FUNCTION_BLOCK booleanAssertionTests EXTENDS FB_TestSuite

VAR
	concrete	: IAssertionTestable;
END_VAR

testBoolIsTrue();
testBoolIsFalse();
testBoolIsEqual();
testBoolIsNotEqual();

METHOD FB_init : BOOL
VAR_INPUT
    bInitRetains : BOOL; // if TRUE, the retain variables are initialized (warm start / cold start)
    bInCopyCode : BOOL;  // if TRUE, the instance afterwards gets moved into the copy code (online change)
	concrete : IAssertionTestable;
END_VAR
THIS^.concrete := concrete;
END_METHOD

METHOD reset
VAR_INPUT
END_VAR
THIS^.concrete.assertionWasWrong  := FALSE;
END_METHOD

METHOD testBoolIsEqual

VAR
	testVarCurrent : BOOL;
	testVarExpected : BOOL;
END_VAR
TEST('Boolean is EqualTo' );

// Test Number 0
THIS^.reset();
THIS^.concrete.assert.boolean.valueIsEqualTo(
	currentValue 	:= testVarCurrent,
	expectedValue	:= testVarExpected,
	message			:= ''
);

THIS^.AssertEquals_BOOL(
	Expected 	:= FALSE,
	Actual 		:= THIS^.concrete.assertionWasWrong,
	Message 	:= 'Test number 0 for boolean.isEqualTo assertion failed'
);

// Test Number 1
THIS^.reset();
testVarCurrent := TRUE;
THIS^.concrete.assert.boolean.valueIsEqualTo(
	currentValue 	:= testVarCurrent,
	expectedValue	:= testVarExpected,
	message			:= ''
);

THIS^.AssertEquals_BOOL(
	Expected 	:= TRUE,
	Actual 		:= THIS^.concrete.assertionWasWrong,
	Message 	:= 'Test number 1 for boolean.isEqualTo assertion failed'
);

// Test Number 2
THIS^.reset();
testVarCurrent := FALSE;
testVarExpected := TRUE;
THIS^.concrete.assert.boolean.valueIsEqualTo(
	currentValue 	:= testVarCurrent,
	expectedValue	:= testVarExpected,
	message			:= ''
);

THIS^.AssertEquals_BOOL(
	Expected 	:= TRUE,
	Actual 		:= THIS^.concrete.assertionWasWrong,
	Message 	:= 'Test number 2 for boolean.isEqualTo assertion failed'
);

// Test Number 3
THIS^.reset();
testVarCurrent := TRUE;
testVarExpected := FALSE;
THIS^.concrete.assert.boolean.valueIsEqualTo(
	currentValue 	:= testVarCurrent,
	expectedValue	:= testVarExpected,
	message			:= ''
);

THIS^.AssertEquals_BOOL(
	Expected 	:= TRUE,
	Actual 		:= THIS^.concrete.assertionWasWrong,
	Message 	:= 'Test number 3 for boolean.isEqualTo assertion failed'
);

// Test Number 4
THIS^.reset();
testVarCurrent := TRUE;
testVarExpected := 0;
THIS^.concrete.assert.boolean.valueIsEqualTo(
	currentValue 	:= testVarCurrent,
	expectedValue	:= testVarExpected,
	message			:= ''
);

THIS^.AssertEquals_BOOL(
	Expected 	:= TRUE,
	Actual 		:= THIS^.concrete.assertionWasWrong,
	Message 	:= 'Test number 4 for boolean.isEqualTo assertion failed'
);

// Test Number 5
THIS^.reset();
testVarCurrent := 1;
testVarExpected := 0;
THIS^.concrete.assert.boolean.valueIsEqualTo(
	currentValue 	:= testVarCurrent,
	expectedValue	:= testVarExpected,
	message			:= ''
);

THIS^.AssertEquals_BOOL(
	Expected 	:= TRUE,
	Actual 		:= THIS^.concrete.assertionWasWrong,
	Message 	:= 'Test number 5 for boolean.isEqualTo assertion failed'
);

// Test Number 6
THIS^.reset();
testVarCurrent := 1;
testVarExpected := 1;
THIS^.concrete.assert.boolean.valueIsEqualTo(
	currentValue 	:= testVarCurrent,
	expectedValue	:= testVarExpected,
	message			:= ''
);

THIS^.AssertEquals_BOOL(
	Expected 	:= FALSE,
	Actual 		:= THIS^.concrete.assertionWasWrong,
	Message 	:= 'Test number 6 for boolean.isEqualTo assertion failed'
);

// Test Number 7
THIS^.reset();
testVarCurrent := 0;
testVarExpected := 0;
THIS^.concrete.assert.boolean.valueIsEqualTo(
	currentValue 	:= testVarCurrent,
	expectedValue	:= testVarExpected,
	message			:= ''
);

THIS^.AssertEquals_BOOL(
	Expected 	:= FALSE,
	Actual 		:= THIS^.concrete.assertionWasWrong,
	Message 	:= 'Test number 7 for boolean.isEqualTo assertion failed'
);

// Test Number 8
THIS^.reset();
testVarCurrent := TRUE;
testVarExpected := TRUE;
THIS^.concrete.assert.boolean.valueIsEqualTo(
	currentValue 	:= testVarCurrent,
	expectedValue	:= testVarExpected,
	message			:= ''
);

THIS^.AssertEquals_BOOL(
	Expected 	:= FALSE,
	Actual 		:= THIS^.concrete.assertionWasWrong,
	Message 	:= 'Test number 8 for boolean.isEqualTo assertion failed'
);

// Test Number 9
THIS^.reset();
testVarCurrent := FALSE;
testVarExpected := FALSE;
THIS^.concrete.assert.boolean.valueIsEqualTo(
	currentValue 	:= testVarCurrent,
	expectedValue	:= testVarExpected,
	message			:= ''
);

THIS^.AssertEquals_BOOL(
	Expected 	:= FALSE,
	Actual 		:= THIS^.concrete.assertionWasWrong,
	Message 	:= 'Test number 9 for boolean.isEqualTo assertion failed'
);

TEST_FINISHED();
END_METHOD

METHOD testBoolIsFalse

VAR
	testBoolVar : BOOL;	
END_VAR
TEST('Boolean is False' );

// Test number 0
THIS^.reset();
THIS^.concrete.assert.boolean.valueIsFalse(
	currentValue 	:= testBoolVar,
	message			:= ''
);						

THIS^.AssertEquals_BOOL(
	Expected 	:= FALSE,
	Actual 		:= THIS^.concrete.assertionWasWrong,
	Message 	:= 'Test number 0 for boolean.isFalse assertion failed'
);

// Test number 1
THIS^.reset();
testBoolVar := TRUE;
THIS^.concrete.assert.boolean.valueIsFalse(
	currentValue 	:= testBoolVar,
	message			:= ''
);						

THIS^.AssertEquals_BOOL(
	Expected 	:= TRUE,
	Actual 		:= THIS^.concrete.assertionWasWrong,
	Message 	:= 'Test number 1 for boolean.isFalse assertion failed'
);

// Test number 2
THIS^.reset();
testBoolVar := FALSE;
THIS^.concrete.assert.boolean.valueIsFalse(
	currentValue 	:= testBoolVar,
	message			:= ''
);						

THIS^.AssertEquals_BOOL(
	Expected 	:= FALSE,
	Actual 		:= THIS^.concrete.assertionWasWrong,
	Message 	:= 'Test number 2 for boolean.isFalse assertion failed'
);

// Test number 3
THIS^.reset();
testBoolVar := 0;
THIS^.concrete.assert.boolean.valueIsFalse(
	currentValue 	:= testBoolVar,
	message			:= ''
);						

THIS^.AssertEquals_BOOL(
	Expected 	:= FALSE,
	Actual 		:= THIS^.concrete.assertionWasWrong,
	Message 	:= 'Test number 3 for boolean.isFalse assertion failed'
);

// Test number 4
THIS^.reset();
testBoolVar := 1;
THIS^.concrete.assert.boolean.valueIsFalse(
	currentValue 	:= testBoolVar,
	message			:= ''
);						

THIS^.AssertEquals_BOOL(
	Expected 	:= TRUE,
	Actual 		:= THIS^.concrete.assertionWasWrong,
	Message 	:= 'Test number 4 for boolean.isFalse assertion failed'
);
TEST_FINISHED();
END_METHOD

METHOD testBoolIsNotEqual

VAR
	testVarCurrent : BOOL;
	testVarExpected : BOOL;
END_VAR
TEST('Boolean is NotEqualTo' );

// Test Number 0
THIS^.reset();
THIS^.concrete.assert.boolean.valueIsNotEqualTo(
	currentValue 	:= testVarCurrent,
	unexpectedValue	:= testVarExpected,
	message			:= ''
);

THIS^.AssertEquals_BOOL(
	Expected 	:= TRUE,
	Actual 		:= THIS^.concrete.assertionWasWrong,
	Message 	:= 'Test number 0 for boolean.notEqualTo assertion failed'
);

// Test Number 1
THIS^.reset();
testVarCurrent := TRUE;
THIS^.concrete.assert.boolean.valueIsNotEqualTo(
	currentValue 	:= testVarCurrent,
	unexpectedValue	:= testVarExpected,
	message			:= ''
);

THIS^.AssertEquals_BOOL(
	Expected 	:= FALSE,
	Actual 		:= THIS^.concrete.assertionWasWrong,
	Message 	:= 'Test number 1 for boolean.notEqualTo assertion failed'
);

// Test Number 2
THIS^.reset();
testVarCurrent := FALSE;
testVarExpected := TRUE;
THIS^.concrete.assert.boolean.valueIsNotEqualTo(
	currentValue 	:= testVarCurrent,
	unexpectedValue	:= testVarExpected,
	message			:= ''
);

THIS^.AssertEquals_BOOL(
	Expected 	:= FALSE,
	Actual 		:= THIS^.concrete.assertionWasWrong,
	Message 	:= 'Test number 2 for boolean.notEqualTo assertion failed'
);

// Test Number 3
THIS^.reset();
testVarCurrent := TRUE;
testVarExpected := FALSE;
THIS^.concrete.assert.boolean.valueIsNotEqualTo(
	currentValue 	:= testVarCurrent,
	unexpectedValue	:= testVarExpected,
	message			:= ''
);

THIS^.AssertEquals_BOOL(
	Expected 	:= FALSE,
	Actual 		:= THIS^.concrete.assertionWasWrong,
	Message 	:= 'Test number 3 for boolean.notEqualTo assertion failed'
);

// Test Number 4
THIS^.reset();
testVarCurrent := TRUE;
testVarExpected := 0;
THIS^.concrete.assert.boolean.valueIsNotEqualTo(
	currentValue 	:= testVarCurrent,
	unexpectedValue	:= testVarExpected,
	message			:= ''
);

THIS^.AssertEquals_BOOL(
	Expected 	:= FALSE,
	Actual 		:= THIS^.concrete.assertionWasWrong,
	Message 	:= 'Test number 4 for boolean.notEqualTo assertion failed'
);

// Test Number 5
THIS^.reset();
testVarCurrent := 1;
testVarExpected := 0;
THIS^.concrete.assert.boolean.valueIsNotEqualTo(
	currentValue 	:= testVarCurrent,
	unexpectedValue	:= testVarExpected,
	message			:= ''
);

THIS^.AssertEquals_BOOL(
	Expected 	:= FALSE,
	Actual 		:= THIS^.concrete.assertionWasWrong,
	Message 	:= 'Test number 5 for boolean.notEqualTo assertion failed'
);

// Test Number 6
THIS^.reset();
testVarCurrent := 1;
testVarExpected := 1;
THIS^.concrete.assert.boolean.valueIsNotEqualTo(
	currentValue 	:= testVarCurrent,
	unexpectedValue	:= testVarExpected,
	message			:= ''
);

THIS^.AssertEquals_BOOL(
	Expected 	:= TRUE,
	Actual 		:= THIS^.concrete.assertionWasWrong,
	Message 	:= 'Test number 6 for boolean.notEqualTo assertion failed'
);

// Test Number 7
THIS^.reset();
testVarCurrent := 0;
testVarExpected := 0;
THIS^.concrete.assert.boolean.valueIsNotEqualTo(
	currentValue 	:= testVarCurrent,
	unexpectedValue	:= testVarExpected,
	message			:= ''
);

THIS^.AssertEquals_BOOL(
	Expected 	:= TRUE,
	Actual 		:= THIS^.concrete.assertionWasWrong,
	Message 	:= 'Test number 7 for boolean.notEqualTo assertion failed'
);

// Test Number 8
THIS^.reset();
testVarCurrent := TRUE;
testVarExpected := TRUE;
THIS^.concrete.assert.boolean.valueIsNotEqualTo(
	currentValue 	:= testVarCurrent,
	unexpectedValue	:= testVarExpected,
	message			:= ''
);

THIS^.AssertEquals_BOOL(
	Expected 	:= TRUE,
	Actual 		:= THIS^.concrete.assertionWasWrong,
	Message 	:= 'Test number 8 for boolean.notEqualTo assertion failed'
);

// Test Number 9
THIS^.reset();
testVarCurrent := FALSE;
testVarExpected := FALSE;
THIS^.concrete.assert.boolean.valueIsNotEqualTo(
	currentValue 	:= testVarCurrent,
	unexpectedValue	:= testVarExpected,
	message			:= ''
);

THIS^.AssertEquals_BOOL(
	Expected 	:= TRUE,
	Actual 		:= THIS^.concrete.assertionWasWrong,
	Message 	:= 'Test number 9 for boolean.notEqualTo assertion failed'
);

TEST_FINISHED();
END_METHOD

METHOD testBoolIsTrue

VAR
	testBoolVar : BOOL;	
END_VAR
TEST('Boolean is true' );

// Test number 0
THIS^.reset();
THIS^.concrete.assert.boolean.valueIsTrue(
	currentValue 	:= testBoolVar,
	message			:= ''
);						

THIS^.AssertEquals_BOOL(
	Expected 	:= TRUE,
	Actual 		:= THIS^.concrete.assertionWasWrong,
	Message 	:= 'Test number 0 for boolean.isTrue assertion failed'
);

// Test number 1
THIS^.reset();
testBoolVar := TRUE;
THIS^.concrete.assert.boolean.valueIsTrue(
	currentValue 	:= testBoolVar,
	message			:= ''
);						

THIS^.AssertEquals_BOOL(
	Expected 	:= FALSE,
	Actual 		:= THIS^.concrete.assertionWasWrong,
	Message 	:= 'Test number 1 for boolean.isTrue assertion failed'
);

// Test number 2
THIS^.reset();
testBoolVar := FALSE;
THIS^.concrete.assert.boolean.valueIsTrue(
	currentValue 	:= testBoolVar,
	message			:= ''
);						

THIS^.AssertEquals_BOOL(
	Expected 	:= TRUE,
	Actual 		:= THIS^.concrete.assertionWasWrong,
	Message 	:= 'Test number 2 for boolean.isTrue assertion failed'
);

// Test number 3
THIS^.reset();
testBoolVar := 0;
THIS^.concrete.assert.boolean.valueIsTrue(
	currentValue 	:= testBoolVar,
	message			:= ''
);						

THIS^.AssertEquals_BOOL(
	Expected 	:= TRUE,
	Actual 		:= THIS^.concrete.assertionWasWrong,
	Message 	:= 'Test number 3 for boolean.isTrue assertion failed'
);

// Test number 4
THIS^.reset();
testBoolVar := 1;
THIS^.concrete.assert.boolean.valueIsTrue(
	currentValue 	:= testBoolVar,
	message			:= ''
);						

THIS^.AssertEquals_BOOL(
	Expected 	:= FALSE,
	Actual 		:= THIS^.concrete.assertionWasWrong,
	Message 	:= 'Test number 4 for boolean.isTrue assertion failed'
);
TEST_FINISHED();
END_METHOD

END_FUNCTION_BLOCK

(* stored: Version 1.1.0.1, ProductVersion 3.1.4024.10
   POU booleanAssertionTests: Id {fd06dce1-b875-4eda-bbe4-1c666534cc7d}, SpecialFunc None
   Method FB_init: Id {7607b5b1-6ade-4578-804a-1a62b0dfa64b}
   Method reset: Id {ba5f2b27-beb3-4d42-8e5e-40348a957cfc}
   Method testBoolIsEqual: Id {a421e08f-2bb3-4e58-9238-320fa7938001}
   Method testBoolIsFalse: Id {233a94f4-fc7b-4644-8b34-b7584775243f}
   Method testBoolIsNotEqual: Id {480da3e2-de0c-4630-943b-cdbbe348c796}
   Method testBoolIsTrue: Id {2e7a1f02-7e27-47aa-8f26-834d914775bb} *)
